FUNCTION_BLOCK KickoutStation EXTENDS MachineStation
VAR_INPUT
	rIO					: REFERENCE TO Kickout_IO_typ;
	rStation			: REFERENCE TO Station;
	rOrientStation 		: REFERENCE TO Station;
	rTrayLoadStation	: REFERENCE TO MultiStation;

END_VAR
VAR_OUTPUT
END_VAR
VAR
	Payload			: Payload_typ;
END_VAR

IF NOT (__ISVALIDREF(rStation) AND __ISVALIDREF(rIO) AND __ISVALIDREF(rOrientStation) ) THEN
	ADSLOGSTR( ADSLOG_MSGTYPE_ERROR, 'Invalid reference at %s.', InstancePath);	// how to make this work?
	RETURN;
END_IF

IF Enable THEN
	IF NOT _Enable THEN
		;
	END_IF

	CASE State OF
		STN_WAIT:
			IF Run AND rStation.MoverInPosition THEN
				State	:= STN_CHECKMOVER;
				Payload	:= rStation.CurrentMover.Payload;
			END_IF

		STN_CHECKMOVER:
			
		IF rIO.Inputs.BallRemoved THEN 
			// Oops ??
		ELSE
			rIO.Outputs.BallClampOpen := TRUE;
			State := STN_OPENBALLCLAMP;
				
		END_IF
			
		
		STN_OPENBALLCLAMP:
			IF rIO.Inputs.BallClampOpened THEN
				rIO.Outputs.BallClampOpen	:= FALSE;
				rIO.Outputs.RemoveBall		:= TRUE;
				State						:= STN_PROCESS;
			END_IF

		STN_PROCESS:
			IF rIO.Inputs.BallRemoved THEN
				rIO.Outputs.RemoveBall		:= FALSE;
				Payload.HasBall 			:= FALSE;
				Payload.BallSeated 			:= FALSE;
				Payload.Reject 				:= FALSE;
				rIO.Outputs.BallClampClose 	:= TRUE;
				State 						:= STN_CLOSEBALLCLAMP;
			END_IF;
			
		STN_CLOSEBALLCLAMP:
			IF rIO.Inputs.BallClampClosed THEN
				rIO.Outputs.BallClampClose 	:= FALSE;
				State						:= STN_SEND;
			END_IF

		STN_SEND:

			rStation.CurrentMover.Payload	:= Payload;
			rStation.CurrentMover.MoveToMultiStation(rTrayLoadStation);
			rStation.CurrentMover.MoveToStation(rOrientStation);
			rStation.UnregisterCurrent();

			State							:= STN_WAIT;
		
		STN_ERROR:
	
	END_CASE

ELSIF _Enable THEN
	rIO.Outputs.BallClampClose	:= FALSE;
	rIO.Outputs.BallClampOpen	:= FALSE;
	rIO.Outputs.RemoveBall		:= FALSE;
	State	:= STN_WAIT;
END_IF

//Save Previous Values
_Enable	:= Enable;

END_FUNCTION_BLOCK

(* stored: Version 1.1.0.1, ProductVersion 3.1.4024.12
   POU KickoutStation: Id {1842ff95-20fa-0ac9-39e6-1dfcb969a2fa}, SpecialFunc None *)
